# EPICS autosave request: calc/calcApp/Db/userCalcOuts10_settings.req
file calcout_settings.req P=$(P)userCalcOut1
file calcout_settings.req P=$(P)userCalcOut2
file calcout_settings.req P=$(P)userCalcOut3
file calcout_settings.req P=$(P)userCalcOut4
file calcout_settings.req P=$(P)userCalcOut5
file calcout_settings.req P=$(P)userCalcOut6
file calcout_settings.req P=$(P)userCalcOut7
file calcout_settings.req P=$(P)userCalcOut8
file calcout_settings.req P=$(P)userCalcOut9
file calcout_settings.req P=$(P)userCalcOut10
